(* IEC 61131-3 sources: teller/JD_Teller_LC2_V11/Class/SIMPULSJE_Teller, 1 file *)

(* ---- SIMPULSJE_Teller.st ---- *)
(*!
<Class
	Name               = "SIMPULSJE_Teller"
	Revision           = "1.0"
	RealtimeTask       = "false"
	CyclicTask         = "true"
	DefCyclictime      = "10 ms"
	BackgroundTask     = "false"
	Sigmatek           = "false"
	OSInterface        = "false"
	HighPriority       = "false"
	Automatic          = "false"
	UpdateMode         = "Prescan"
	SharedCommandTable = "true"
	Objectsize         = "(284,120)">
	<Channels>
		<Server Name="ClassSvr" Visualized="false" Initialize="false" WriteProtected="true" Retentive="false"/>
		<Server Name="SignAaninMs" Visualized="false" Initialize="false" WriteProtected="false" Retentive="false"/>
		<Server Name="SignUitinMs" Visualized="false" Initialize="false" WriteProtected="false" Retentive="false"/>
		<Server Name="TaskOnOff" Visualized="false" Initialize="false" WriteProtected="false" Retentive="false"/>
		<Server Name="Uitgang" Visualized="false" Initialize="false" WriteProtected="true" Retentive="false"/>
	</Channels>
	<RevDoku>
		<Owner Company="JD" Author="SV"/>
		<Dokumentation Revision="1.0" Date="2014-09-23" Author="SV" Company="JD" Description="Kopie van SIMPULSJE. TaskOnOff in init op 1 gezet."/>
	</RevDoku>
</Class>
*)
SIMPULSJE_Teller : CLASS
  //Servers:
	ClassSvr 	: SvrChCmd_DINT;
	TaskOnOff 	: SvrCh_DINT;
	Uitgang 	: SvrCh_DINT;
	SignAaninMs 	: SvrCh_UDINT;
	SignUitinMs 	: SvrCh_UDINT;
  //Clients:
  //Variables:
		timer1 	: DINT;
		timer2 	: UDINT;
		timer3 	: UDINT;
		timer4 	: UDINT;
  //Functions:

	FUNCTION VIRTUAL GLOBAL Init;

	FUNCTION VIRTUAL GLOBAL CyWork
		VAR_INPUT
			EAX 	: UDINT;
		END_VAR
		VAR_OUTPUT
			state (EAX) 	: UDINT;
		END_VAR;

	FUNCTION VIRTUAL GLOBAL RtWork
		VAR_INPUT
			EAX 	: UDINT;
		END_VAR
		VAR_OUTPUT
			state (EAX) 	: UDINT;
		END_VAR;
  //Tables:
	FUNCTION @STD
		VAR_OUTPUT
			ret_code	: CONFSTATES;
		END_VAR;
	FUNCTION GLOBAL TAB @CT_;
END_CLASS;

FUNCTION VIRTUAL GLOBAL SIMPULSJE_Teller::Init

timer1:=0;
SignAaninMs:=250;
SignAaninMs.Write(input:=SignAaninMs);
SignUitinMs:=500;
SignUitinMs.Write(input:=SignUitinMs);

if TaskOnOff = 0 then
 TaskOnOff :=1;
end_if;

END_FUNCTION

FUNCTION VIRTUAL GLOBAL SIMPULSJE_Teller::CyWork
	VAR_INPUT
		EAX 	: UDINT;
	END_VAR
	VAR_OUTPUT
		state (EAX) 	: UDINT;
	END_VAR

//Als in de machine setup de functie is geselelecteerd wordt de code uitgevoerd
  if  TaskOnOff then

      case timer1 of

      0:

            timer2:=ops.tAbsolute;
            timer1+=1;
            Uitgang:=1;
            Uitgang.Write(Uitgang);
      1:

            if (ops.tAbsolute - timer2) > SignAaninMs then
            timer1+=1;
            end_if;

      2:
            timer2:=ops.tAbsolute;
            timer1+=1;
            Uitgang:=0;
            Uitgang.Write(Uitgang);

      3:

            if (ops.tAbsolute-timer2) > SignuitinMs then
            timer1:=0;
            end_if;

      end_case;

  end_if;

	state := READY;

END_FUNCTION

FUNCTION VIRTUAL GLOBAL SIMPULSJE_Teller::RtWork
	VAR_INPUT
		EAX 	: UDINT;
	END_VAR
	VAR_OUTPUT
		state (EAX) 	: UDINT;
	END_VAR

	state := READY;

END_FUNCTION
